{attribute addProperty BoxType "EL3312-0000-0016"}
{attribute addProperty Id "TC_Inputs_ChannelAT %I*ARRAY[0..8] OF TC_Inputs_Channel_E5019A8F144180WcStateAT %I*WcState_98A4DF7520.250InfoDataAT %I*InfoData_BC63D37F80100"}
{attribute addProperty CRC "121607544"}
{attribute addProperty SizeInBites "226"}
{attribute addProperty SizeInBytes "28.25"}
TYPE EL3312_4A09AC12 :
STRUCT
	{attribute addProperty Name "TC_Inputs_Channel"}
	TC_Inputs_Channel : ARRAY[0..8] OF TC_Inputs_Channel_E5019A8F;
	{attribute addProperty Name "WcState"}
	WcState : WcState_98A4DF75;
	{attribute addProperty Name "InfoData"}
	InfoData : InfoData_BC63D37F;
END_STRUCT
END_TYPE

(* stored: Version 1.2.0.0, ProductVersion 3.1.4024.9
   DUT EL3312_4A09AC12: Id {ffb57d75-1f5e-4138-aee5-d6474fdaf852} *)
